TYPE T_OUTER_Barcode : T_MaxString;
END_TYPE

(* stored: Version 1.1.0.1
   DUT T_OUTER_Barcode: Id {be2669ae-6a81-49c8-897a-1e12b8e467fb} *)
